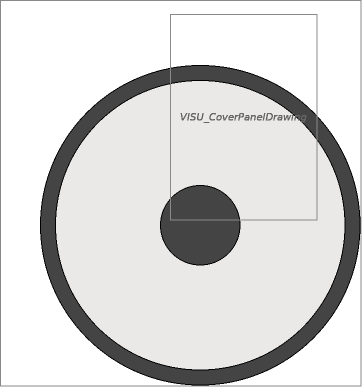
VISUALIZATION VISU_CoverPanelOverviewDrawing  // 362x387
VAR_IN_OUT
	cover : Cover;
	coverWidget : CoverWidget;	
END_VAR
    Ellipse (40,65 320x320)
    Ellipse (55,80 290x290)
    Ellipse (160,185 80x80)
    Frame (170,14 147x206)
        shows VISU_CoverPanelDrawing(coverPanelConfig := cover.config.top.p1, coverPanel := cover.parts.top.parts.p1, widget := coverWidget.top.p1)
    Frame (170,14 147x206)
        shows VISU_CoverPanelDrawing(coverPanelConfig := cover.config.bottom.p1, coverPanel := cover.parts.bottom.parts.p1, widget := coverWidget.bottom.p1)
    Frame (170,14 147x206)
        shows VISU_CoverPanelDrawing(coverPanelConfig := cover.config.top.p2, coverPanel := cover.parts.top.parts.p2, widget := coverWidget.top.p2)
    Frame (170,14 147x206)
        shows VISU_CoverPanelDrawing(coverPanelConfig := cover.config.bottom.p2, coverPanel := cover.parts.bottom.parts.p2, widget := coverWidget.bottom.p2)
    Frame (170,14 147x206)
        shows VISU_CoverPanelDrawing(coverPanelConfig := cover.config.top.p3, coverPanel := cover.parts.top.parts.p3, widget := coverWidget.top.p3)
    Frame (170,14 147x206)
        shows VISU_CoverPanelDrawing(coverPanelConfig := cover.config.bottom.p3, coverPanel := cover.parts.bottom.parts.p3, widget := coverWidget.bottom.p3)
    Frame (170,14 147x206)
        shows VISU_CoverPanelDrawing(coverPanelConfig := cover.config.top.p4, coverPanel := cover.parts.top.parts.p4, widget := coverWidget.top.p4)
    Frame (170,14 147x206)
        shows VISU_CoverPanelDrawing(coverPanelConfig := cover.config.bottom.p4, coverPanel := cover.parts.bottom.parts.p4, widget := coverWidget.bottom.p4)
END_VISUALIZATION

(* stored: Version 1.1.0.1, ProductVersion 3.1.4019.2
   Visu VISU_CoverPanelOverviewDrawing: Id {4fbdc7e5-dbdc-4540-9711-7625730f553a} *)
